Fanuc KAREL source: ks00035.KL

-- PROVISIONAL review KL for V1013-1; original PC SHA256 d8afeac036652511bd6bed970455617401d42f513e0d4f2763588f88416a405b
-- Incomplete behavior may be omitted. Consult companion uncertainty JSON. Do not deploy.
PROGRAM KS00035
%NOLOCKGROUP
VAR
  FLAG : BOOLEAN
  N : INTEGER
  STATUS : INTEGER
  PN : STRING[80]
  VN : STRING[80]
-- UNRESOLVED_DECL A type=00201c
-- UNRESOLVED_DECL B type=00201c
BEGIN
  -- UNRESOLVED_PC offsets 5-13; opcodes 3F,75
  -- UNRESOLVED_PC offsets 18-27; opcodes 3F,75
  -- UNRESOLVED_PC offsets 32-70; opcodes 27,22,22,2A,22,2A,22,22,B0
  -- UNRESOLVED_PC offsets 75-79; opcodes 7F
END KS00035
